PROGRAM MAIN
VAR
Xas: AXIS_REF;
Yas: AXIS_REF;

XMotorPower: MC_power; 
YMotorPower: MC_power;
XMotorPosition: MC_MoveAbsolute;
YMotorPosition: MC_MoveAbsolute;
XMotorHome: MC_Home;
YMotorHome: MC_Home;
Estop AT %I*: BOOL;
links: BOOL;
rechts: BOOL;
XMotorReset: MC_Reset;
YMotorReset: MC_Reset;

END_VAR

//Deze code is gemaakt om te testen hoe een servomotor moest worden aangestuurd. Deze code is niet actief betrokken in de huidige plc code.

XMotorPosition(Axis := Xas, Velocity := 250, Acceleration := 10, Deceleration := 2000, Jerk := 100000);
YMotorPosition(Axis := Yas, Velocity := 250, Acceleration := 10, Deceleration := 2000, Jerk := 100000);
XMotorPower(Axis:= Xas, Enable := TRUE, Enable_Positive := TRUE, Enable_Negative := TRUE);
YMotorPower(Axis:= Yas, Enable := TRUE, Enable_Positive := TRUE, Enable_Negative := TRUE);


//XMotorHome(Axis := Xas, Execute := TRUE, Position := 0, HomingMode := MC_DIRECT); 

IF links AND NOT rechts AND Estop THEN
	XMotorPosition(Axis := Xas, Execute := TRUE, Position:= 500);
END_IF

IF NOT links AND rechts AND Estop THEN
	XMotorPosition(Axis := Xas, Execute := TRUE, Position:= -500);
END_IF

IF NOT Estop THEN
	XMotorPosition( Axis := Xas, Execute := FALSE);
END_IF

END_PROGRAM

(* stored: Version 1.1.0.1, ProductVersion 3.1.4024.12
   POU MAIN: Id {c9b5f613-7e3f-4340-8405-66d9cf0a3910}, SpecialFunc None *)
